// TwinCAT 3 PLC project Main
// ProgramVersion: 3.1.4023.0
// libraries:
//   mobject-json, * (mobject.io)
//   Tc2_Standard, * (Beckhoff Automation GmbH)
//   Tc2_System, * (Beckhoff Automation GmbH)
//   Tc3_Module, * (Beckhoff Automation GmbH)
//   TcUnit, * (www.tcunit.org)
// project tree:
//   / PlcTask.TcTTO
//   POUs/ MAIN.TcPOU
//   Tests/ JsonPath_TestSuit.TcPOU, TEST_PRG.TcPOU
// real-time tasks:
//   TASK PlcTask: cycle T#10ms, priority 20, ADS port 350

CONFIGURATION Main
    RESOURCE PLC ON TwinCAT3
        TASK PlcTask(INTERVAL := T#10ms, PRIORITY := 20);
        PROGRAM MAIN WITH PlcTask : MAIN;
    END_RESOURCE
END_CONFIGURATION

// ---- POUs/MAIN.TcPOU
PROGRAM MAIN
VAR
	
	jsonPath : JsonPath;
	json : T_MAXSTRING := '{"factory":{"machines":[{"name":"module 1","in-production":true,"speed":122.2,"produced":608},{"name":"module 2","in-production":false,"speed":543.2,"produced":24}]}}';

	machineName : STRING;
	inProduction : BOOL;
	speed : LREAL;
	produced : INT;
	myInt : INT;
	
	hresult : HRESULT;
	
END_VAR

// setup the json reader with the supplied json

jsonPath.Parse(json);

// all paths are found and can be automatically converted to the supplied destination variables

hresult := jsonPath.TryRead('factory.machines[0].name',machineName); // hresult = S_OK, machineName = 'module 1'
hresult := jsonPath.TryRead('.factory.machines[0].in-production',inProduction); // hresult = S_OK, inProduction = true
hresult := jsonPath.TryRead('$$factory.machines[1].speed',speed); // hresult = S_OK, speed = 543.2
hresult := jsonPath.TryRead('$$.[$'factory$'].machines[1].produced',produced); // hresult = S_OK, produced = 24

// this will fail as 122.2 cannot be automatically converted to the type INT without data loss. 

hresult := jsonPath.TryRead('.factory.machines[0].speed',myInt); // hresult = INCOMPATIBLE, myInt = no change

// this will fail as the property 'hello' cannot be found. 

hresult := jsonPath.TryRead('.factory.machines[0].hello',myInt); // hresult = NOTFOUND, myInt = no change

// library test runner
TEST_PRG();

END_PROGRAM

// ---- Tests/TEST_PRG.TcPOU
PROGRAM TEST_PRG
VAR
	jsonPath_Test : JsonPath_TestSuit;
END_VAR

jsonPath_Test();

TcUnit.RUN();

END_PROGRAM

// ---- Tests/JsonPath_TestSuit.TcPOU
FUNCTION_BLOCK JsonPath_TestSuit EXTENDS TcUnit.FB_TestSuite
VAR
	jsonPath : JsonPath;
END_VAR

ReadBoolFromJsonString();
ReadIntFromJsonString();
ReadDIntFromJsonString();
ReadUDIntFromJsonString();
ReadRealFromJsonString();
ReadLRealFromJsonString();
ReadStringFromJsonString();

METHOD PUBLIC ReadBoolFromJsonString
VAR_INPUT
END_VAR
VAR
	jsonTestString : T_MAXSTRING := '{"myTrueBool" : true, "myFalseBool" : false}';
	trueBool : BOOL := FALSE;
	falseBOOL : BOOL := TRUE;
END_VAR
TEST('ReadBoolFromJsonString');

// @TEST-RUN
jsonPath.Parse(jsonTestString);
jsonPath.TryRead('.myTrueBool',trueBool);
jsonPath.TryRead('.myFalseBool',falseBool);

// @TEST-ASSERT
AssertTrue(Condition := trueBool, Message := 'jsonPath read boolean did not read true');
AssertFalse(Condition := falseBool, Message := 'jsonPath read boolean did not read false');

TEST_FINISHED();
END_METHOD

METHOD PUBLIC ReadDIntFromJsonString
VAR_INPUT
END_VAR
VAR
	jsonTestString : T_MAXSTRING := '{"myDInt" : 123}';
	Actual : DINT;
	Expected : DINT := 123;
END_VAR
TEST('ReadDIntFromJsonString');

// @TEST-RUN
jsonPath.Parse(jsonTestString);
jsonPath.TryRead('.myDInt',Actual);

// @TEST-ASSERT
AssertEquals(Expected := Expected, Actual := Actual, Message := 'jsonPath did not read correct value');

TEST_FINISHED();
END_METHOD

METHOD PUBLIC ReadIntFromJsonString
VAR_INPUT
END_VAR
VAR
	jsonTestString : T_MAXSTRING := '{"myInt" : 123}';
	Actual : INT;
	Expected : INT := 123;
END_VAR
TEST('ReadIntFromJsonString');

// @TEST-RUN
jsonPath.Parse(jsonTestString);
jsonPath.TryRead('.myInt',Actual);

// @TEST-ASSERT
AssertEquals(Expected := Expected, Actual := Actual, Message := 'jsonPath did not read correct value');

TEST_FINISHED();
END_METHOD

METHOD PUBLIC ReadLRealFromJsonString
VAR_INPUT
END_VAR
VAR
	jsonTestString : T_MAXSTRING := '{"myLReal" : -123.1}';
	Actual : LREAL;
	Expected : LREAL := -123.1;
END_VAR
TEST('ReadLRealFromJsonString');

// @TEST-RUN
jsonPath.Parse(jsonTestString);
jsonPath.TryRead('.myLReal',Actual);

// @TEST-ASSERT
AssertEquals(Expected := Expected, Actual := Actual, Message := 'jsonPath did not read correct value');

TEST_FINISHED();
END_METHOD

METHOD PUBLIC ReadRealFromJsonString
VAR_INPUT
END_VAR
VAR
	jsonTestString : T_MAXSTRING := '{"myReal" : 123.1}';
	Actual : REAL;
	Expected : REAL := 123.1;
END_VAR
TEST('ReadRealFromJsonString');

// @TEST-RUN
jsonPath.Parse(jsonTestString);
jsonPath.TryRead('.myReal',Actual);

// @TEST-ASSERT
AssertEquals(Expected := Expected, Actual := Actual, Message := 'jsonPath did not read correct value');

TEST_FINISHED();
END_METHOD

METHOD PUBLIC ReadStringFromJsonString
VAR_INPUT
END_VAR
VAR
	jsonTestString : T_MAXSTRING := '{"myString" : "test"}';
	Actual : T_MAXSTRING;
	Expected : T_MAXSTRING := 'test';
END_VAR
TEST('ReadStringFromJsonString');

// @TEST-RUN
jsonPath.Parse(jsonTestString);
jsonPath.TryRead('.myString',Actual);

// @TEST-ASSERT
AssertEquals(Expected := Expected, Actual := Actual, Message := 'jsonPath did not read correct value');

TEST_FINISHED();
END_METHOD

METHOD PUBLIC ReadUDIntFromJsonString
VAR_INPUT
END_VAR
VAR
	jsonTestString : T_MAXSTRING := '{"myUDInt" : 123}';
	Actual : UDINT;
	Expected : UDINT := 123;
END_VAR
TEST('ReadUDIntFromJsonString');

// @TEST-RUN
jsonPath.Parse(jsonTestString);
jsonPath.TryRead('.myUDInt',Actual);

// @TEST-ASSERT
AssertEquals(Expected := Expected, Actual := Actual, Message := 'jsonPath did not read correct value');

TEST_FINISHED();
END_METHOD

END_FUNCTION_BLOCK
